{attribute 'qualified_only'}
{attribute 'strict'}
TYPE E_ModuleSequenceCommand :
(
	Begin,
	Block,
	Resume,
	Cancel,
	Reiterate,
	Revert	
);
END_TYPE

(* stored: Version 1.1.0.1, ProductVersion 3.1.4024.9
   DUT E_ModuleSequenceCommand: Id {eb3d6b49-adde-47fa-9770-5fb2e21c491d} *)
